{attribute 'qualified_only'}
{attribute 'strict'}
TYPE E_Timer :
(
	Timer0 := 0,
	Line0PriorityOnDelay,     // 主流线优先置位延时
	Line0PriorityOffDelay,    // 主流线优先复位延时
	SteeringCheck1F,
	OpenLockCheckF,
	Timer5,
	Timer6,
	Timer7,
	Timer8,
	Timer9,
	Timer10,
	Timer11,
	Timer12,
	Timer13,
	Timer14,
	Timer15,
	Timer16,
	Timer17,
	Timer18,
	Timer19
	
);
END_TYPE

(* stored: Version 1.1.0.1, ProductVersion 3.1.4024.3
   EnumerationTextList E_Timer: Id {eb662605-a822-47ab-9c44-16b2cc4dae4e} *)
